INTERFACE ITF_BaseGroupElement_HMI_Connector_View EXTENDS ITF_BaseControlElement_HMI_Connector_View

END_INTERFACE

(* stored: Version 1.1.0.1
   Itf ITF_BaseGroupElement_HMI_Connector_View: Id {886a85bc-d9f2-0b34-350a-7828be6ba314} *)
